PROGRAM MAIN
VAR
	//tank : tank1;
	//tank : Tank1_1;
	tank : Tank1_1_1;
	bfill : BOOL;
 
END_VAR


tank(bSwitchFill := bfill);

END_PROGRAM

(* stored: Version 1.1.0.1, ProductVersion 3.1.4024.0
   POU MAIN: Id {5923207b-7a28-40c0-bfea-04bf7407582a}, SpecialFunc None *)
